// TIA Portal project "PLCII_Pro1" (V15.1)

(* hardware
DEVICE "S7-1200 station_1"  S7-1200 Station
   slot 0: "Rack_0"  S7-1200 Rack  Rack  V1.0
   slot 1: "PLC_1"  CPU 1215C AC/DC/Rly  6ES7 215-1BG40-0XB0  V4.2
*)

// ===== PLC "PLC_1"  CPU 1215C AC/DC/Rly =====

VAR_GLOBAL   // PLC tag table "Default tag table"
   "Start" AT %M0.0 : Bool;
   "Sys_runing" AT %M0.1 : Bool;
   "Stop" AT %M0.2 : Bool;
   "Tag" AT %M0.3 : Bool;
   "ONST" AT %M0.4 : Bool;
   "activate" AT %M2.5 : Bool;
   "tagi" AT %M0.6 : Bool;
END_VAR

DATA_BLOCK "ReciverSystem"   // DB1
{ S7_Optimized_Access := 'TRUE' }
VERSION : 0.1
   VAR
      PressureLevel : Int;
      SW_90PSI : Bool;
      SW_110PSI : Bool;
      Pump : Bool;
      Light : Bool;
      Level_State : Int;
      System_State : Int;
   END_VAR
BEGIN
END_DATA_BLOCK

DATA_BLOCK "PressureTest_DB"   // DB2
{ S7_Optimized_Access := 'TRUE' }
VERSION : 0.1
// stored: InstanceOfName PressureTest
"PressureTest"
BEGIN
END_DATA_BLOCK

FUNCTION_BLOCK "PressureTest"   // FB1, LAD
{ S7_Optimized_Access := 'TRUE' }
VERSION : 0.1
   VAR
      ONS1 : Bool;
      ONS2 : Bool;
      Sys_activated : Bool;
   END_VAR
   VAR_TEMP   // added for the SCL form of the ladder/FBD networks
      _w1 : Bool;
      _w2 : Bool;
   END_VAR
BEGIN

REGION Network 1
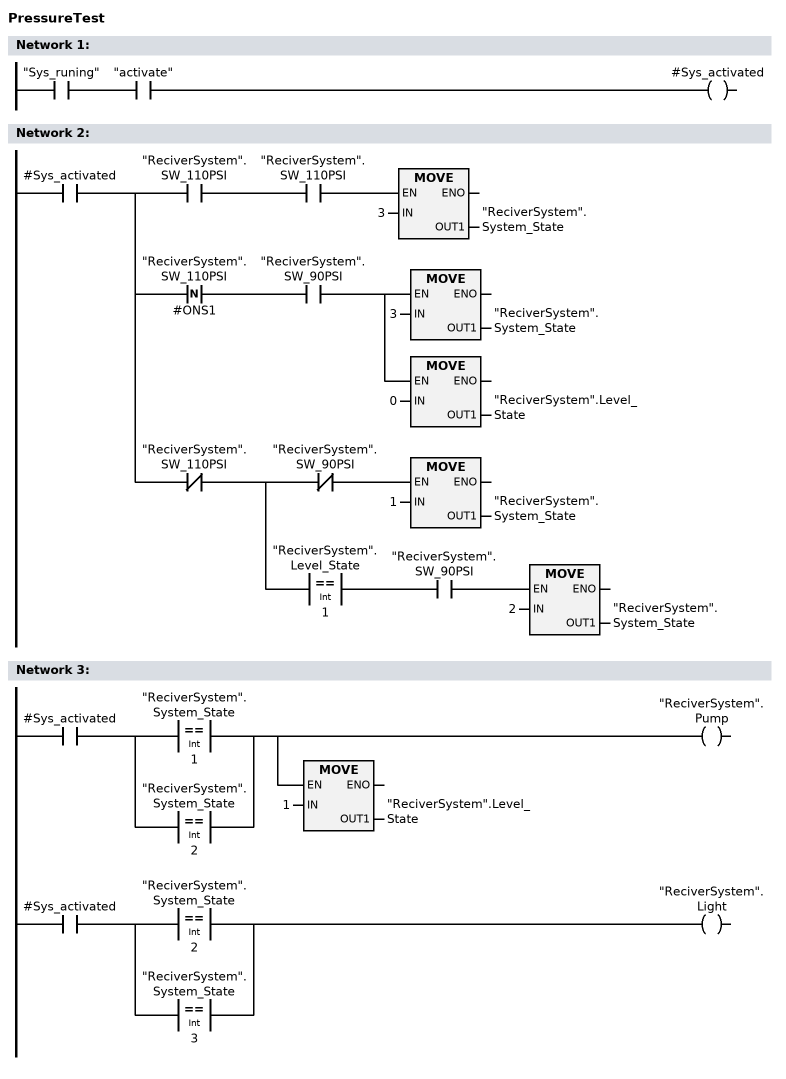
   RUNG wire#powerrail
      Contact( "Sys_runing" )
      Contact( "activate" )
      Coil( #Sys_activated )
   END_RUNG
   // the same network as SCL:
   #Sys_activated := "Sys_runing" AND "activate";
END_REGION

REGION Network 2
   RUNG wire#powerrail
      Contact( #Sys_activated )
      wire#w1
      Contact( "ReciverSystem".SW_110PSI )
      Contact( "ReciverSystem".SW_110PSI )
      Move(in := 3, out1 => "ReciverSystem".System_State)
   END_RUNG
   RUNG wire#w1
      N_Contact(operand := "ReciverSystem".SW_110PSI, bit := #ONS1)
      Contact( "ReciverSystem".SW_90PSI )
      wire#w2
      Move(in := 3, out1 => "ReciverSystem".System_State)
   END_RUNG
   RUNG wire#w2
      Move(in := 0, out1 => "ReciverSystem".Level_State)
   END_RUNG
   RUNG wire#w1
      I_Contact( "ReciverSystem".SW_110PSI )
      wire#w3
      I_Contact( "ReciverSystem".SW_90PSI )
      Move(in := 1, out1 => "ReciverSystem".System_State)
   END_RUNG
   RUNG wire#w3
      { S7_Templates := "SrcType := Int" } EQ_Contact(in1 := "ReciverSystem".Level_State, in2 := 1)
      Contact( "ReciverSystem".SW_90PSI )
      Move(in := 2, out1 => "ReciverSystem".System_State)
   END_RUNG
   // the same network as SCL:
   IF #Sys_activated AND "ReciverSystem".SW_110PSI AND "ReciverSystem".SW_110PSI THEN
       "ReciverSystem".System_State := 3;
   END_IF;
   #_w1 := #Sys_activated AND NOT "ReciverSystem".SW_110PSI AND #ONS1;   // falling edge of "ReciverSystem".SW_110PSI
   #ONS1 := "ReciverSystem".SW_110PSI;
   IF #_w1 AND "ReciverSystem".SW_90PSI THEN
       "ReciverSystem".System_State := 3;
       "ReciverSystem".Level_State := 0;
   END_IF;
   #_w2 := #Sys_activated AND NOT "ReciverSystem".SW_110PSI;
   IF #_w2 AND NOT "ReciverSystem".SW_90PSI THEN "ReciverSystem".System_State := 1; END_IF;
   IF #_w2 AND ("ReciverSystem".Level_State = 1) AND "ReciverSystem".SW_90PSI THEN
       "ReciverSystem".System_State := 2;
   END_IF;
END_REGION

REGION Network 3
   RUNG wire#powerrail
      Contact( #Sys_activated )
      wire#w1
      { S7_Templates := "SrcType := Int" } EQ_Contact(in1 := "ReciverSystem".System_State, in2 := 1)
      wire#w2
      Coil( "ReciverSystem".Pump )
   END_RUNG
   RUNG wire#w1
      { S7_Templates := "SrcType := Int" } EQ_Contact(in1 := "ReciverSystem".System_State, in2 := 2)
   END_RUNG wire#w2
   RUNG wire#w2
      Move(in := 1, out1 => "ReciverSystem".Level_State)
   END_RUNG
   RUNG wire#powerrail
      Contact( #Sys_activated )
      wire#w3
      { S7_Templates := "SrcType := Int" } EQ_Contact(in1 := "ReciverSystem".System_State, in2 := 2)
      wire#w4
      Coil( "ReciverSystem".Light )
   END_RUNG
   RUNG wire#w3
      { S7_Templates := "SrcType := Int" } EQ_Contact(in1 := "ReciverSystem".System_State, in2 := 3)
   END_RUNG wire#w4
   // the same network as SCL:
   "ReciverSystem".Pump := #Sys_activated AND (("ReciverSystem".System_State = 1) OR ("ReciverSystem".System_State = 2));
   IF "ReciverSystem".Pump THEN "ReciverSystem".Level_State := 1; END_IF;
   "ReciverSystem".Light := #Sys_activated AND (("ReciverSystem".System_State = 2) OR ("ReciverSystem".System_State = 3));
END_REGION
END_FUNCTION_BLOCK

ORGANIZATION_BLOCK "OB_cycle"   // OB1, LAD, ProgramCycle
TITLE = "Main Program Sweep (Cycle)"
{ S7_Optimized_Access := 'TRUE' }
VERSION : 0.1
   VAR_INPUT
      Initial_Call : Bool;   // Initial call of this OB
      Remanence : Bool;   // =True, if remanent data are available
   END_VAR
   VAR_TEMP   // added for the SCL form of the ladder/FBD networks
      _w1 : Bool;
   END_VAR
BEGIN

REGION Network 1
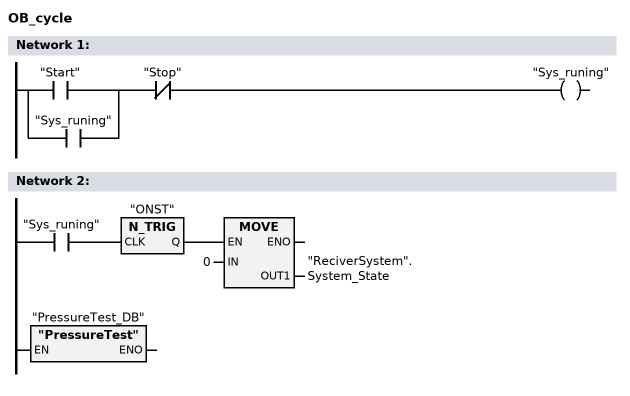
   RUNG wire#powerrail
      Contact( "Start" )
      wire#w1
      I_Contact( "Stop" )
      Coil( "Sys_runing" )
   END_RUNG
   RUNG wire#powerrail
      Contact( "Sys_runing" )
   END_RUNG wire#w1
   // the same network as SCL:
   "Sys_runing" := ("Start" OR "Sys_runing") AND NOT "Stop";
END_REGION

REGION Network 2
   RUNG wire#powerrail
      Contact( "Sys_runing" )
      N_Trig( "ONST" )
      Move(in := 0, out1 => "ReciverSystem".System_State)
   END_RUNG
   RUNG wire#powerrail
      "PressureTest_DB"()
   END_RUNG
   // the same network as SCL:
   #_w1 := NOT "Sys_runing" AND "ONST";   // falling edge
   "ONST" := "Sys_runing";
   IF #_w1 THEN "ReciverSystem".System_State := 0; END_IF;
   "PressureTest_DB"();   // "PressureTest"
END_REGION
END_ORGANIZATION_BLOCK